# EPICS autosave request: iocBoot/iocvxWorks/interp_settings.req
$(P)interp.A
$(P)interp.B
$(P)interp.C
$(P)interp.E
$(P)interp.F
$(P)interp_y1.DESC
$(P)interp_y2.DESC
$(P)interp_y1.OUT
$(P)interp_y2.OUT
